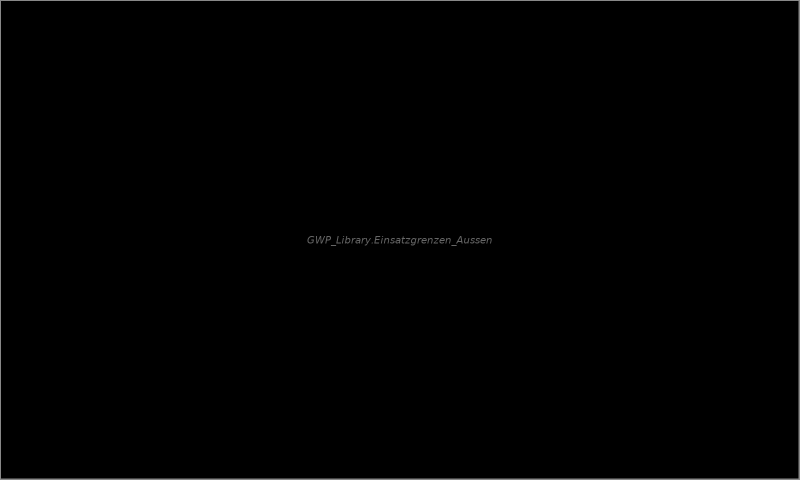
VISUALIZATION EG_Aussen  // 800x480
    Frame (0,0 800x480)
        shows GWP_Library.Einsatzgrenzen_Aussen(FB_Einsatzgrenzen_Aussen := Main.Einsatzgrenzen_Aussen_0, FB_Init_1 := Main.Init_0)
END_VISUALIZATION

(* stored: Version 1.1.0.1, ProductVersion 3.1.4022.6
   Visu EG_Aussen: Id {8621bf4f-6429-49d4-bdf9-70faa706ec1f} *)
